{attribute addProperty BoxType "EJ1957-0000-0017"}
{attribute addProperty Id "Channel_1_Standard_OutputAT %Q*BOOL811Channel_2_Standard_OutputAT %Q*BOOL812Channel_3_Standard_OutputAT %Q*BOOL813Channel_4_Standard_OutputAT %Q*BOOL814"}
{attribute addProperty CRC "851047905"}
{attribute addProperty SizeInBites "32"}
{attribute addProperty SizeInBytes "4"}
TYPE Outputs_32B9F5E1 :
STRUCT
	{attribute addProperty Name "Channel_1_Standard_Output"}
	Channel_1_Standard_Output AT %Q* : BOOL;
	{attribute addProperty Name "Channel_2_Standard_Output"}
	Channel_2_Standard_Output AT %Q* : BOOL;
	{attribute addProperty Name "Channel_3_Standard_Output"}
	Channel_3_Standard_Output AT %Q* : BOOL;
	{attribute addProperty Name "Channel_4_Standard_Output"}
	Channel_4_Standard_Output AT %Q* : BOOL;
END_STRUCT
END_TYPE

(* stored: Version 1.2.0.0, ProductVersion 3.1.4024.9
   DUT Outputs_32B9F5E1: Id {f94f2e0f-c25f-41b9-9717-c2d3f252f9f6} *)
